TYPE AutoCtrlCmds :
STRUCT
	Start: BOOL;
	Stop: BOOL;
	Emergency: BOOL;
	Reset: BOOL;
	
	ProcessReady: BOOL;
	ProcessRun: BOOL;
	ProcessFault: BOOL;
END_STRUCT
END_TYPE

(* stored: Version 1.1.0.1, ProductVersion 3.1.4024.4
   DUT AutoCtrlCmds: Id {403ac9ea-31e2-4ebe-b815-e3db0e06f0bd} *)
